FUNCTION_BLOCK FB_Mover IMPLEMENTS IMover
VAR
	axesEnable		: MC_Power;
	axesReset		: AxesReset(_axis);
	axesMoveTo 		: MoveMoverToPosition(_axis) := (Gap := 100.0);
	axesHalt 		: HaltMover(_axis);
	axesReadError : Tc2_MC2.MC_ReadAxisError;
	_axis 			: AXIS_REF;
	_identInGroup : INT;
	_trackLength : MC_LREAL;
	_targetPos : LREAL;
	_MoverErrorId : DWORD;
	_arrZones : ARRAY[1..4] OF DINT;
	_arrVelocities : ARRAY[1..4] OF mc_LREAL;
END_VAR

axesMoveTo();
axesHalt();
axesReset();
_axis.ReadStatus();
axesEnable(Axis := _axis);
axesReadError(Axis := _axis, Enable := TRUE, AxisErrorID => _MoverErrorId);

PROPERTY PUBLIC Acceleration : mc_lreal
GET
Acceleration := axesMoveTo.Acceleration;
END_GET
SET
axesMoveTo.Acceleration := Acceleration;
END_SET
END_PROPERTY

PROPERTY PUBLIC AxisRef : reference to AXIS_REF
GET
AxisRef REF= THIS^._axis;
END_GET
END_PROPERTY

PROPERTY PUBLIC Deceleration : mc_lreal
GET
Deceleration := axesMoveTo.Deceleration;
END_GET
SET
axesMoveTo.Deceleration := Deceleration;
END_SET
END_PROPERTY

METHOD PUBLIC DisableAxis : BOOL
VAR_INPUT
END_VAR
axesEnable.Enable := false;
END_METHOD

METHOD PUBLIC EnableAxis : BOOL
VAR_INPUT
END_VAR
axesEnable.Enable := axesEnable.Enable_Negative := axesEnable.Enable_Positive := TRUE;
axesEnable.Override := 100;
END_METHOD

PROPERTY PUBLIC Gap : mc_lreal
GET
Gap := axesMoveTo.Gap;
END_GET
SET
axesMoveTo.Gap := Gap;
END_SET
END_PROPERTY

METHOD PUBLIC HaltAxis : BOOL
VAR_INPUT
END_VAR
IF NOT axesHalt.Busy THEN
	axesHalt.Execute();
	HaltAxis := TRUE;
	axesMoveTo.Abort();
END_IF
END_METHOD

METHOD PUBLIC HasCommand : BOOL
VAR_INPUT
END_VAR
HasCommand := axesMoveTo.Busy;
END_METHOD

METHOD hasError : BOOL
VAR_INPUT
END_VAR
hasError := _axis.Status.Error;
END_METHOD

PROPERTY PUBLIC IdentInGroup : int
GET
IdentInGroup := _identInGroup;
END_GET
SET
_identInGroup := IdentInGroup;
END_SET
END_PROPERTY

METHOD isAtPosition : BOOL
VAR_INPUT
	position : MC_LREAL;
END_VAR
IF position > 1 THEN
	IF _axis.NcToPlc.ModuloActPos < position + 1 AND _axis.NcToPlc.ModuloActPos > position - 1 THEN
		isAtPosition := TRUE;
	END_IF  
ELSE
	IF _axis.NcToPlc.ModuloActPos < position + 1 AND _axis.NcToPlc.ModuloActPos > 0.0  
		OR _axis.NcToPlc.ModuloActPos < _trackLength AND _axis.NcToPlc.ModuloActPos > _trackLength - 1 THEN
		isAtPosition := TRUE;
	END_IF
END_IF
END_METHOD

METHOD PUBLIC isDetected : BOOL
VAR_INPUT
END_VAR
IF _axis.NcToPlc.AxisId = 0 THEN
	RETURN;
END_IF
isDetected := true;
END_METHOD

METHOD isEnabled : BOOL
VAR_INPUT
END_VAR
isEnabled := not _axis.Status.Disabled;
END_METHOD

METHOD PUBLIC isPastPosition : BOOL
VAR_INPUT
	position : MC_LREAL;
END_VAR
IF position > 1 THEN
	IF _axis.NcToPlc.ModuloActPos > position THEN
		isPastPosition := TRUE;
	END_IF  
END_IF
END_METHOD

METHOD PUBLIC isStationary : BOOL
VAR_INPUT
END_VAR
isStationary := _axis.NcToPlc.SetVelo = 0;
END_METHOD

PROPERTY PUBLIC Jerk : mc_lreal
GET
Jerk := axesMoveTo.Jerk;
END_GET
SET
axesMoveTo.Jerk := Jerk;
END_SET
END_PROPERTY

METHOD PROTECTED ModuloToAbs : mc_lreal
VAR_INPUT
	moduloPositionDemand: MC_LREAL;
	_backwardsAllowed : BOOL;
END_VAR
//---------code to set actual position from modulo command----------------------
IF NOT _backwardsAllowed THEN
	//--------if you want to go forward-------------------------------------------------------------
	//---------if SetPos is greater than current actual then move to that position--------------------
	//---------else current position is greater, increase moduloturn count by 1 before set---------------
	IF moduloPositionDemand > _axis.NcToPlc.ModuloActPos THEN
		ModuloToAbs := (DINT_TO_LREAL(_Axis.NcToPlc.ModuloActTurns)*_trackLength) + moduloPositionDemand;
	ELSE
		ModuloToAbs := (DINT_TO_LREAL(_Axis.NcToPlc.ModuloActTurns + 1)*_trackLength) + moduloPositionDemand;
	END_IF
ELSE
	//--------if you want to go backwards--------------------------------
	//--------if setPos is less than current actual then move to that position---------------------
	//---------else current position is less, decrease moduloturn count by 1 before set------------
	IF moduloPositionDemand < _axis.NcToPlc.ModuloActPos THEN
		ModuloToAbs := (DINT_TO_LREAL(_Axis.NcToPlc.ModuloActTurns)*_trackLength) + moduloPositionDemand;
	ELSE
		ModuloToAbs := (DINT_TO_LREAL(_Axis.NcToPlc.ModuloActTurns-1)*_trackLength) + moduloPositionDemand;
	END_IF
END_IF
END_METHOD

PROPERTY MoverErrorId : dword
GET
MoverErrorId := _MoverErrorId;
END_GET
SET
_MoverErrorId := MoverErrorId;
END_SET
END_PROPERTY

METHOD PUBLIC MoveTo : BOOL
VAR_INPUT
	Position : MC_LREAL;
	Velocity : MC_LREAL;
	BackwardMove : BOOL;
END_VAR
IF NOT isAtPosition(position := Position) THEN
	IF NOT axesMoveTo.Busy THEN
		axesMoveTo.MoveTo(Position := ModuloToAbs(Position, BackwardMove), Velocity := Velocity);
		MoveTo := TRUE;
		_targetPos := Position;
	END_IF
END_IF
END_METHOD

METHOD PUBLIC ResetAxis : BOOL
VAR_INPUT
END_VAR
VAR
END_VAR
axesReset.Execute();
axesMoveTo.Abort();
axesHalt.Abort();
END_METHOD

PROPERTY PUBLIC TrackLength : MC_LREAL
GET
TrackLength := _trackLength;
END_GET
SET
_trackLength := TrackLength;
END_SET
END_PROPERTY

PROPERTY Zones : array[1..4] of dint
GET
Zones := _arrZones;
END_GET
SET
_arrZones := Zones;
END_SET
END_PROPERTY

PROPERTY ZoneVelocities : array[1..4] of mc_lreal
GET
ZoneVelocities := _arrVelocities;
END_GET
SET
_arrVelocities := ZoneVelocities;
END_SET
END_PROPERTY

END_FUNCTION_BLOCK

(* stored: Version 1.1.0.1, ProductVersion 3.1.4024.12
   POU FB_Mover: Id {85f62a02-889f-4b30-9036-53b84a79c2ee}, SpecialFunc None
   Folder Methods: Id {d990f5ad-a7ee-4f95-bbee-90adbd32272b}
   Folder Properties: Id {9a91c5be-52fe-48a0-bc15-6ebc4b6012ce}
   Property Acceleration: Id {a3bda034-ea93-4d84-971d-34fbe2eb3e0f}
   Get Get: Id {8c0c7777-8a58-44b5-831c-d4a0cf61096f}
   Set Set: Id {15b9d915-5373-4e6e-a7cf-25aa0d155d51}
   Property AxisRef: Id {2843dfe6-0082-40ff-8e1b-e945b442209e}
   Get Get: Id {441b4e2d-2dd8-4dfd-acba-52c3ad9f53ca}
   Property Deceleration: Id {00007a36-41b4-4823-a8e6-8b128b9220ef}
   Get Get: Id {0743f223-d07f-40e0-ae56-9ad8fd39c497}
   Set Set: Id {8a8da0aa-4ad5-4681-8cbf-8df29be399b8}
   Method DisableAxis: Id {04391d47-2802-4391-8e85-6f6f9a8009c0}
   Method EnableAxis: Id {916b8003-bdc6-4d15-969b-eb3f20546af3}
   Property Gap: Id {df4301cc-49ae-42f0-9fb5-132b4f344460}
   Get Get: Id {b3b25d73-9e78-4a8e-aa02-29541270bc33}
   Set Set: Id {1ed6cdb7-78d2-4469-8882-1352cf35da3a}
   Method HaltAxis: Id {5275c1d7-51e4-468b-bae6-7d197b328c9f}
   Method HasCommand: Id {844de5ea-f5c0-4a84-91ef-26224d069b5b}
   Method hasError: Id {0731dcbf-a6a0-405e-88ac-62fdc749ce1d}
   Property IdentInGroup: Id {863b9761-cbc8-44d8-8050-2a1636e9b23e}
   Get Get: Id {2460ad73-8e3d-445e-b8d7-9b894aa7ea8e}
   Set Set: Id {69a139ab-9ae0-43c6-b9bf-2377ec4e46f3}
   Method isAtPosition: Id {67155926-7eff-4cd8-a436-a6125aa63be5}
   Method isDetected: Id {1c403adf-75d5-4d1d-b5e5-98c1b51f5e05}
   Method isEnabled: Id {fae51c40-d1bc-41c8-b30b-e977362b0398}
   Method isPastPosition: Id {e98ee30c-01c3-4bc5-a45f-19f156a6d04e}
   Method isStationary: Id {cc970b73-1098-42f9-b684-982f1c612571}
   Property Jerk: Id {9a69768d-c95b-4d14-9731-0ca2801ab119}
   Get Get: Id {9e7bb0c7-f81a-4b2b-b010-20db407de009}
   Set Set: Id {1d8fcd9c-d31e-49a8-abee-3c36b6c0dd41}
   Method ModuloToAbs: Id {1ab38b34-3edf-4bf3-ac63-8f2c352a45b5}
   Property MoverErrorId: Id {2137719e-b5a1-4682-a2d0-0001ce8d8ee5}
   Get Get: Id {1b6a7ee9-2942-41cf-9596-83f1f808cbe8}
   Set Set: Id {1d09e392-50e7-4b60-8ed6-6bb0b4703e36}
   Method MoveTo: Id {72bb7891-d6a7-452b-a0d5-5ef44fec51ae}
   Method ResetAxis: Id {39a27677-b6f4-4959-8c10-40191fe8181b}
   Property TrackLength: Id {7929754e-f474-406b-9ccc-2835a01be62c}
   Get Get: Id {74c84618-ed54-44f2-8255-e9174e3733ee}
   Set Set: Id {65927336-9892-421b-815d-67d2ffb9474c}
   Property Zones: Id {7132752b-9f59-4a46-a150-43ba47619df1}
   Get Get: Id {75ce3c1d-eb75-4217-9e15-d93820df891e}
   Set Set: Id {e14ede83-145e-4ae1-b1a2-80b0712b7280}
   Property ZoneVelocities: Id {0c9eec13-62ea-46e0-bfc7-5fba619d4227}
   Get Get: Id {a716ace3-ff6d-43c7-b98d-4fb9e88f4e04}
   Set Set: Id {4bccd87c-6aff-47f6-b004-f22954a42a30} *)
